(* PLC project LibIT, lamsystems-it.ru LibIT 1 *)
(* stored: creationDateTime 2019-11-13T09:37:45, productRelease 0, modificationDateTime 2022-04-28T12:46:30, version 0 *)

(* Increment of source value *)
FUNCTION Inc : INT
  VAR_INPUT
    Ex : BOOL;  (* execution allow *)
    V : INT;  (* source value *)
  END_VAR
  VAR
    Val : INT;
  END_VAR

            Val:= V;

IF Ex = True THEN
  Val:= V+1;
END_IF;

Inc:= Val;


          
END_FUNCTION

(* Decrement of source value *)
FUNCTION Dec : INT
  VAR_INPUT
    Ex : BOOL;  (* execution allow *)
    V : INT;  (* source value *)
  END_VAR
  VAR
    Val : INT;
  END_VAR

            Val:= V;

IF Ex = True AND Val > 0 THEN
  Val:= V-1;
END_IF;

Dec:= Val;


          
END_FUNCTION

(* Set bit value in source word *)
FUNCTION SetBitLWo : LWORD
  VAR_INPUT
    Wo : LWORD := 0;  (* source word *)
    Pos : BYTE := 0;  (* bit position (0..63) *)
    Val : BOOL := FALSE;  (* bit value *)
  END_VAR
  VAR
    Mask : LWORD := 0;
  END_VAR

            Mask:= REAL_TO_LWORD(EXPT(INT_TO_REAL(2),BYTE_TO_INT(Pos)));
IF Val = FALSE THEN
  SetBitLWo:= (Wo AND NOT(Mask));
ELSE
  SetBitLWo:= (Wo OR Mask);
END_IF;
          
END_FUNCTION

(* Get bit value from source word *)
FUNCTION GetBitLWo : BOOL
  VAR_INPUT
    Wo : LWORD := 0;  (* source word *)
    Pos : BYTE := 0;  (* bit position (0..63) *)
  END_VAR
  VAR
    Mask : LWORD := 0;
  END_VAR

            Mask:= REAL_TO_LWORD(EXPT(INT_TO_REAL(2),BYTE_TO_INT(Pos)));
GetBitLWo:= ((Wo AND Mask) > 0);

          
END_FUNCTION

(* Set bit value in source word *)
FUNCTION SetBitWo : WORD
  VAR_INPUT
    Wo : WORD := 0;  (* source word *)
    Pos : BYTE := 0;  (* bit position (0..15) *)
    Val : BOOL := FALSE;  (* bit value *)
  END_VAR
  VAR
    Mask : WORD := 0;
  END_VAR

            Mask:= REAL_TO_WORD(EXPT(INT_TO_REAL(2),BYTE_TO_INT(Pos)));
IF Val = FALSE THEN
  SetBitWo:= (Wo AND NOT(Mask));
ELSE
  SetBitWo:= (Wo OR Mask);
END_IF;
          
END_FUNCTION

(* Get bit value from source word *)
FUNCTION GetBitWo : BOOL
  VAR_INPUT
    Wo : WORD := 0;  (* source word *)
    Pos : BYTE := 0;  (* bit position (0..15) *)
  END_VAR
  VAR
    Mask : WORD := 0;
  END_VAR

            Mask:= REAL_TO_WORD(EXPT(INT_TO_REAL(2),BYTE_TO_INT(Pos)));
GetBitWo:= ((Wo AND Mask) > 0);

          
END_FUNCTION

(* Filtration of discrete value *)
FUNCTION_BLOCK FiltrD
  VAR_INPUT
    Ex : BOOL := FALSE;  (* execution allow *)
    V : BOOL := FALSE;  (* source value *)
    Tm : TIME := T#0ms;  (* filter delay (ms) *)
  END_VAR
  VAR_OUTPUT
    Ov : BOOL := FALSE;  (* filtered source value *)
  END_VAR
  VAR
    Val : BOOL := FALSE;
    TON0 : TON;
    TON1 : TON;
  END_VAR

            TON0(IN:=AND(Ex, NOT(V)), PT:=Tm);
TON1(IN:=AND(Ex, V), PT:=Tm);

IF TON0.Q = TRUE THEN
  Val:= FALSE;
END_IF;

IF TON1.Q = TRUE THEN
  Val:= TRUE;
END_IF;

Ov:= Val;

          
END_FUNCTION_BLOCK

(* Filtration of analog value *)
FUNCTION_BLOCK FiltrA
  VAR_INPUT
    Ex : BOOL := FALSE;  (* execution allow *)
    V : REAL := 0.0;  (* source value *)
    K : REAL := 0.0;  (* filter factor (0.0 .. 1.0) *)
  END_VAR
  VAR_OUTPUT
    Ov : REAL := 0.0;  (* filtered source value *)
  END_VAR
  VAR
    Val : REAL := 0.0;  (* stored value *)
    Klim : REAL := 0.0;  (* stored value *)
  END_VAR

            IF Ex = TRUE THEN
  Klim:= LIMIT(MN:=0.0, IN:=K, MX:=1.0);
  Val := (Klim*V)+(1.0-Klim)*Ov;
ELSE
  Val:= V;
END_IF;

Ov:= Val;

          
END_FUNCTION_BLOCK

(* Calculate scale angle factor *)
FUNCTION ScaleA_Ka : REAL
  VAR_INPUT
    Ex : BOOL := FALSE;  (* execution allow *)
    V1 : REAL := 0.0;  (* value of low point *)
    V2 : REAL := 0.0;  (* value of high point *)
    Y1 : REAL := 0.0;  (* calibration value of low point *)
    Y2 : REAL := 0.0;  (* calibration value of high point *)
    Ka : REAL := 0.0;  (* source value of the factor *)
  END_VAR

            IF Ex = TRUE THEN
  ScaleA_Ka:= (Y2-Y1)/(V2-V1);
ELSE  
  ScaleA_Ka:= Ka;
END_IF;

          
END_FUNCTION

(* Calculate scale offset factor *)
FUNCTION ScaleA_Kb : REAL
  VAR_INPUT
    Ex : BOOL := FALSE;  (* execution allow *)
    V1 : REAL := 0.0;  (* value of low point *)
    V2 : REAL := 0.0;  (* value of high point *)
    Y1 : REAL := 0.0;  (* calibration value of low point *)
    Y2 : REAL := 0.0;  (* calibration value of high point *)
    Kb : REAL := 0.0;  (* source value of the factor *)
  END_VAR

            IF Ex = TRUE THEN
  ScaleA_Kb:= ((Y1*V2)-(Y2*V1))/(V2-V1);
ELSE  
  ScaleA_Kb:= Kb;
END_IF;

          
END_FUNCTION

(* Scale of analog value *)
FUNCTION ScaleA : REAL
  VAR_INPUT
    Ex : BOOL := FALSE;  (* execution allow *)
    V : REAL := 0.0;  (* value of curent point *)
    Ka : REAL := 0.0;  (* angle factor *)
    Kb : REAL := 0.0;  (* offset factor *)
    Y : REAL := 0.0;  (* source scale value *)
  END_VAR

            IF Ex = TRUE THEN
  ScaleA:= (Ka*V)+Kb;
ELSE  
  ScaleA:= Y;
END_IF;

          
END_FUNCTION

(* Continuous TON *)
FUNCTION_BLOCK TONcont
  VAR_INPUT
    IN : BOOL := FALSE;  (* start command *)
  END_VAR
  VAR_OUTPUT
    Q : BOOL := FALSE;  (* status *)
    ET : TIME := T#0ms;  (* estimated time *)
  END_VAR
  VAR
    TON1 : TON;
    TON1_IN : BOOL := FALSE;
    TON1_TM : TIME := T#600000ms;
    TON1Inc : TON;
    TON1Inc_IN : BOOL := FALSE;
    TON1Inc_TM : TIME := T#300000ms;
  END_VAR

            TON1_IN   := IN;
TON1Inc_IN:= IN;

IF TON1Inc.Q = TRUE THEN
  TON1_TM   := ADD_TIME(IN1:=TON1_TM, IN2:=TON1Inc_TM);
  TON1Inc_IN:= FALSE;
END_IF;

TON1(IN:=TON1_IN, PT:=TON1_TM);
TON1Inc(IN:=TON1Inc_IN, PT:=TON1Inc_TM);

Q := TON1.Q;
ET:= TON1.ET;

          
END_FUNCTION_BLOCK

(* Autotuning of PID-controller *)
FUNCTION_BLOCK PIDtun
  VAR_INPUT
    Ex : BOOL := FALSE;  (* execution allow *)
    V : REAL := 0.0;  (* source value *)
    Diff : REAL := 0.0;  (* difference setpoint *)
    Ty : BYTE := 0;  (* type of controller *)
    Pro : BYTE := 0;  (* type of process *)
  END_VAR
  VAR_OUTPUT
    Ok : BYTE := 0;  (* result code *)
    OY : REAL := 0.0;  (* regulator value *)
    OKp : REAL := 0.0;  (* P-factor *)
    OKi : REAL := 0.0;  (* I-factor *)
    OKd : REAL := 0.0;  (* D-factor *)
    OTm : DWORD := 0;  (* cycle time (ms) *)
  END_VAR
  VAR
    OTmLocal : DWORD := 0;  (* cycle time (ms) *)
  END_VAR
  VAR_OUTPUT
    dETm : DWORD := 0;  (* error break control time (ms) *)
  END_VAR
  VAR
    dETmLocal : DWORD := 0;  (* error break control time (ms) *)
  END_VAR
  VAR_OUTPUT
    dE : REAL := 0.0;  (* dE value *)
  END_VAR
  VAR
    dELocal : REAL := 0.0;  (* dE value *)
    TunDone : BOOL := FALSE;
    Tm1 : REAL := 0.0;  (* t0 (ms) *)
    Tm2 : REAL := 0.0;  (* tu (ms) *)
    TmSum : REAL := 0.0;  (* t (ms) *)
    V1Set : BOOL := FALSE;
    V01 : REAL := 0.0;
    V063 : REAL := 0.0;
    Rr : REAL := 0.0;  (* R *)
    Tm1sec : REAL := 0.0;  (* t0 div 100 *)
    TONcont1 : TONcont;
    TONcont1_IN : BOOL := FALSE;
    CntChangeInVal : UINT := 0;
    StartVal : REAL := 0.0;
    PrewVal : REAL := 0.0;
  END_VAR

            (* Ty - regulator type *)
(* = 0 - PID *)
(* = 1 - PI *)
(* = 2 - PD *)
(* = 3 - P *)

(* Pro - process type *)
(* = 0 - increasing (by default) *)
(* = 1 - decreasing *)

(* Ok - result code *)
(* = 0 - off *)
(* = 1 - work *)
(* = 2 - incorrect regulator type *)
(* = 3 - work done success *)

IF Ex = TRUE THEN
  
  IF Ty <= 3 THEN
      
    IF TunDone = FALSE THEN
      
      (* work *)
      Ok:= 1;
      
      IF V1Set = FALSE THEN
        V1Set:= TRUE;
        CntChangeInVal:= 0;
        StartVal:= V;
        PrewVal:= V;        
        (* calculate setpoint for V(0.1) by type of process *)
        IF Pro = 1 THEN
          (* decreasing *)
          V01 := (V-(0.1*Diff));
          V063:= (V-(0.63*Diff));
        ELSE
          (* increasing *)
          V01 := (V+(0.1*Diff));
          V063:= (V+(0.63*Diff));
        END_IF;
      END_IF;
      
      (* set Tm1 (ms) *)
      IF V < V01 THEN
        Tm1:= TIME_TO_REAL(TONcont1.ET)*1000.0;
      END_IF;
      
      (* set Tm2 (ms) *)
      IF V >= V063 THEN
        
        TONcont1_IN:= FALSE;
        TunDone    := TRUE;
        
        Tm2   := TIME_TO_REAL(TONcont1.ET)*1000.0;
        TmSum := (Tm1+Tm2);
        (*OTm   := REAL_TO_DWORD((Tm1*1.875));*)
        Rr    := (Diff/((TmSum-Tm1)/1000.0));
        Tm1sec:= (Tm1/1000.0);
        (* 1000 - divider to convert msec to sec *)
        
        OTm:= OTmLocal; 
        dE:=dELocal;
        dETm:=dETmLocal;                
          
        (* calculate factors by type of regulator *)
        CASE BYTE_TO_INT(Ty) OF
          0:
            (* PID *)
            OKp:= (1.2/(Rr*Tm1sec));
            OKi:= (2.0*Tm1sec);
            OKd:= (0.4*Tm1sec);
          1:
            (* PI *)
            OKp:= (0.8/(Rr*Tm1sec));
            OKi:= (2.0*Tm1sec);
          2:
            (*PD*)
            OKp:= (1.0/(Rr*Tm1sec));
            OKd:= (0.25*Tm1sec);
          3:
            (*P*)
            OKp:= (1.0/(Rr*Tm1sec));
        END_CASE;
        
      END_IF;
      (* end of Tm2 *)
    ELSE
      (* work done success *)
      Ok:= 3;
    END_IF;
    (* end of TunDone *)
  ELSE
    (* incorrect regulator type *)
    Ok:= 2;
  END_IF;
  (* end of Ty *)
ELSE
  (* off *)
  Ok:= 0;
END_IF;
(* end of Ex *)

(* work *)
IF Ok = 1 THEN
  OY         := 100.0;
  TONcont1_IN:= TRUE;
  
  IF CntChangeInVal < 4 THEN  
   IF Pro = 0 THEN (* increasing *)
    IF V > StartVal AND V > PrewVal THEN
      CntChangeInVal:= (CntChangeInVal + 1);
      PrewVal:= V;
    (*ELSE*)
      (*CntChangeInVal:= 0;*)
    END_IF;
   ELSE (* decreasing *)
    IF V < StartVal AND V < PrewVal THEN
      CntChangeInVal:= (CntChangeInVal + 1);
      PrewVal:= V;
    (*ELSE*)
      (*CntChangeInVal:= 0;*)  
    END_IF;   
   END_IF;  
    (*PrewVal:= V;*)  
  END_IF;
  
  IF CntChangeInVal=4 THEN
   OTmLocal:= REAL_TO_DWORD(Tm1); 
   dELocal:=(PrewVal-StartVal);
   dETmLocal:=DINT_TO_DWORD((DWORD_TO_DINT(OTmLocal)*3));
   CntChangeInVal:= 5; 
  END_IF;   
  
END_IF;

(* off, error *)
IF Ok = 0 OR Ok = 2 THEN
  OY         := 0.0;
  TONcont1_IN:= FALSE;
  V1Set      := FALSE;
  TunDone    := FALSE;
  OKp        := 0.0;
  OKi        := 0.0;
  OKd        := 0.0;
  OTm        := 0;
  
  CntChangeInVal:= 0;
  StartVal:= 0.0;
  PrewVal:= 0.0;  
  
  OTmLocal:= 0; 
  dELocal:=0.0;
  dETmLocal:=0;  
  
  OTm:= 0; 
  dE:=0.0;
  dETm:=0;   
  
END_IF;

(* work is done success *)
IF TunDone = TRUE THEN
  OY         := 0.0;
END_IF;

TONcont1(IN:=TONcont1_IN);

(* DEBUG *)
(* set Class of debug variables to Output to use its as Outputs of the FB *)
(* set Class of debug variables to Local to hide its *)
(* Deb_V1 := V01; *)
(* Deb_Tm1:= Tm1; *)
(* Deb_V2 := V063; *)
(* Deb_Tm2:= Tm2; *)
(* end of DEBUG *)

          
END_FUNCTION_BLOCK

(* PID-controller (v1) *)
FUNCTION_BLOCK PID1
  VAR_INPUT
    Ex : BOOL := FALSE;  (* execution allow *)
    V : REAL := 0.0;  (* source value *)
    Sp : REAL := 0.0;  (* setpoint *)
    Ty : BYTE := 0;  (* type of controller *)
    Pro : BYTE := 0;  (* type of process *)
    Kp : REAL := 0.0;  (* P-factor *)
    Ki : REAL := 0.0;  (* I-factor *)
    Kd : REAL := 0.0;  (* D-factor *)
    Sck : BOOL := FALSE;  (* external command to start regulator cycle *)
    dI : REAL := 0.0;  (* integral zone *)
    dZ : REAL := 0.0;  (* dead zone *)
    dE : REAL := 0.0;  (* control failure zone *)
    dETm : DWORD := 5000;  (* control failure zone (time to detect zone, ms) *)
    Ym : BYTE := 0;  (* type of OY *)
  END_VAR
  VAR_OUTPUT
    Ok : BYTE := 0;  (* result code *)
    OY : REAL := 0.0;  (* regulator value (%) *)
  END_VAR
  VAR
    Er : REAL := 0.0;  (* error delta *)
    ErAbs : REAL := 0.0;  (* error delta (absolute) *)
    ErPrev : REAL := 0.0;  (* error delta (previous cycle) *)
    ErDiff : REAL := 0.0;  (* error delta (diff) *)
    Ppart : REAL := 0.0;  (* P-part *)
    Ipart : REAL := 0.0;  (* I-part *)
    Dpart : REAL := 0.0;  (* D-part *)
    DeV : REAL := 0.0;  (* control failure zone (1-point) *)
    DeV1Set : BOOL := FALSE;  (* control failure zone (1-point is set) *)
    DeV2Set : BOOL := FALSE;  (* control failure zone (2-point is set) *)
    SckSet : BOOL := FALSE;  (* external start (set) *)
    ErrorSet : BOOL := FALSE;  (* e-zone (set) *)
    TON_De : TON;
    TON_De_IN : BOOL := FALSE;
    TON_De_TM : TIME := T#0ms;
  END_VAR

            (* Ty - regulator type *)
(* = 0 - PID *)
(* = 1 - PI *)
(* = 2 - PD *)
(* = 3 - P *)

(* Pro - process type *)
(* = 0 - increasing (by default) *)
(* = 1 - decreasing *)

(* Ym - type of OY *)
(* = 0 - unipolar    0.0 .. 100.0 % (by default) *)
(* = 1 - bipolar  -100.0 .. 100.0 % *)

(* Ok - result code *)
(* = 0 - off *)
(* = 1 - work *)
(* = 2 - dead (d-)zone *)
(* = 3 - integral (i-)zone *)
(* = 4 - control failure (e-)zone *)
(* = 5 - incorrect regulator type *)

(* reset Sck *)
IF Sck = FALSE THEN
  SckSet:= FALSE;
END_IF;

(* test execution allow *)
IF Ex = TRUE THEN
  
  (* test regulator type *)
  IF Ty <= 3 THEN
    
    (* test start *)
    IF Sck = TRUE AND SckSet = FALSE AND ErrorSet = FALSE THEN
      
      SckSet:= TRUE;
      
      (* work *)
      Ok:= 1;
     
      Er    := (Sp-V);
      ErDiff:= (Er-ErPrev);
      ErPrev:= Er;
      ErAbs := ABS(IN:=Er);
      
      (* test d-zone *)
      IF ErAbs >= dZ THEN
        
        (* Ty: 0-PID, 1-PI, 2-PD, 3-P *)
        Ppart:= (Kp*Er);
        
        (* Ty: 0-PID, 1-PI *)
        IF (Ty = 0 OR Ty = 1) AND (ErAbs < dI OR dI = 0.0) AND Ki > 0.0 THEN
          (* i-zone *)
          Ok:= 3;
          Ipart:= (Ipart+Er);
          IF Ipart >= Ki THEN
            Ipart:= Ki;
          END_IF;
          Ipart:= ((1.0/Ki)*Ipart);
        ELSE
          Ipart:= 0.0;
        END_IF;
        
        (*0-PID, 2-PD*)
        IF (Ty = 0 OR Ty = 2) THEN
          Dpart:= (Kd*ErDiff);
        ELSE
          Dpart:= 0.0;
        END_IF;
        
        OY:= (Ppart+Ipart+Dpart)*100.0;
        
      ELSE
        (* d-zone *)
        Ok:= 2;
      END_IF;
      (* end of test d-zone *)
      
    END_IF;
    (* end of test start *)
  
  ELSE
    (* incorrect regulator type *)
    Ok:= 5;
    ErrorSet:= TRUE;
  END_IF;
  (* end of test regulator type *)
  
ELSE
  (* off *)
  Ok:= 0;
END_IF;
(* end of Ex *) 

(* work, i-zone *)
IF dETm >= 100 THEN  
 IF (Ok = 1 OR Ok = 3) AND ABS(IN:=OY) >= 100.0 THEN
    
  IF dETm > 0 THEN
    TON_De_TM:= REAL_TO_TIME(DWORD_TO_REAL(dETm)/1000.0);
    TON_De_IN:= TRUE;
  END_IF;
    
  IF DeV1Set = FALSE THEN
    (* point 1 *)
    DeV:= V;
    DeV1Set:= TRUE;
  END_IF;
    
  IF TON_De.Q = TRUE THEN
    IF DeV2Set = FALSE THEN
      (* point 2 *)
      DeV:= (V-DeV);
      DeV2Set:= TRUE;
    END_IF;
    IF DeV < dE OR DeV < 0.0 THEN
      (* e-zone *)
      Ok:= 4;
      ErrorSet:= TRUE;
    END_IF;
  END_IF;
  
 ELSE
  TON_De_IN:= FALSE;
  DeV1Set  := FALSE;
  DeV2Set  := FALSE;
 END_IF;
END_IF;

(* off *)
IF Ok = 0 THEN
  OY       := 0.0;
  SckSet   := FALSE;
  ErrorSet := FALSE;
  Ppart    := 0.0;
  Ipart    := 0.0;
  Dpart    := 0.0;
END_IF;

(* e-zone, error of regulator type *)
IF ErrorSet = TRUE THEN
  OY       := 0.0;
END_IF;

(* scale OY by type of process *)
IF Pro = 1 THEN
  (* decreasing *)
  OY:= (100.0-OY);
END_IF;

(* scale OY by type of output *)
IF Ym = 1 THEN
  (* bipolar *)
  OY:= LIMIT(MN:=-100.0, IN:=OY, MX:=100.0);
ELSE
  (* unipolar *)
  OY:= LIMIT(MN:=0.0, IN:=OY, MX:=100.0);
END_IF;

TON_De(IN:=TON_De_IN, PT:=TON_De_TM);

(* DEBUG *)
(* set Class of debug variables to Output to use its as Outputs of the FB *)
(* set Class of debug variables to Local to hide its *)
(* Deb_P   := Ppart; *)
(* Deb_I   := Ipart; *)
(* Deb_D   := Dpart; *)
(* Deb_dEEt:= REAL_TO_DWORD(TIME_TO_REAL(TON_De.ET)*1000.0); *)
(* end of DEBUG *)

          
END_FUNCTION_BLOCK

(* PID-controller (v2) *)
FUNCTION_BLOCK PID2
  VAR_INPUT
    Ex : BOOL := FALSE;  (* execution allow *)
    V : REAL := 0.0;  (* source value *)
    Sp : REAL := 0.0;  (* setpoint *)
    Ty : BYTE := 0;  (* type of controller *)
    Pro : BYTE := 0;  (* type of process *)
    Kp : REAL := 0.0;  (* P-factor *)
    Ki : REAL := 0.0;  (* I-factor *)
    Kd : REAL := 0.0;  (* D-factor *)
    Tm : DWORD := 1000;  (* cycle time (ms) *)
    dI : REAL := 0.0;  (* integral zone *)
    dZ : REAL := 0.0;  (* dead zone *)
    dE : REAL := 0.0;  (* control failure zone *)
    dETm : DWORD := 5000;  (* control failure zone (time to detect zone, ms) *)
    Ym : BYTE := 0;  (* type of OY *)
  END_VAR
  VAR_OUTPUT
    Ok : BYTE := 0;  (* result code *)
    OY : REAL := 0.0;  (* regulator value (%) *)
  END_VAR
  VAR
    TON_Work : TON;
    TON_Work_IN : BOOL := FALSE;
    TON_Work_TM : TIME := T#0ms;
    PID1_1 : PID1;
  END_VAR

            PID1_1(Ex:=Ex, V:=V, Sp:=Sp, Ty:=Ty, Pro:=Pro, Kp:=Kp, Ki:=Ki, Kd:=Kd, Sck:=TON_Work.Q, dI:=dI, dZ:=dZ, dE:=dE, dETm:=dETm, Ym:=Ym);

Ok:= PID1_1.Ok;
OY:= PID1_1.OY;

IF Ex = TRUE AND Tm > 0 THEN
  TON_Work_TM:= REAL_TO_TIME(DWORD_TO_REAL(Tm)/1000.0);
  TON_Work_IN:= TRUE;
ELSE
  TON_Work_IN:= FALSE;
END_IF;

IF TON_Work.Q = TRUE THEN
  TON_Work_IN:= FALSE;
END_IF;

TON_Work(IN:=TON_Work_IN, PT:=TON_Work_TM);

(* DEBUG *)
(* set Class of debug variables to Output to use its as Outputs of the FB *)
(* set Class of debug variables to Local to hide its *)
(* Deb_P   := PID1_1.Deb_P; *)
(* Deb_I   := PID1_1.Deb_I; *)
(* Deb_D   := PID1_1.Deb_D; *)
(* Deb_Et  := REAL_TO_DWORD(TIME_TO_REAL(TON_Work.ET)*1000.0); *)
(* Deb_dEEt:= PID1_1.Deb_dEEt; *)
(* end of DEBUG *)

          
END_FUNCTION_BLOCK

(* Test TON *)
FUNCTION_BLOCK TONtest
  VAR_INPUT
    IN : BOOL := FALSE;  (* start command *)
    MS : DWORD := 0;  (* counter reference (msec) *)
  END_VAR
  VAR_OUTPUT
    Q : BOOL := FALSE;  (* status *)
    ET : TIME := T#0ms;  (* counter value (msec) *)
    EDW : DWORD := 0;  (* counter value (msec) *)
    EREA : REAL := 0.0;
  END_VAR
  VAR
    TON1 : TON;
    TON1_IN : BOOL := FALSE;
    TON1_TM : TIME := T#0ms;
  END_VAR

            TON1_IN:= IN;
TON1_TM:= REAL_TO_TIME(DWORD_TO_REAL(MS)/1000.0);

TON1(IN:=TON1_IN, PT:=TON1_TM);
Q   := TON1.Q;
ET  := TON1.ET;
EDW := REAL_TO_DWORD(TIME_TO_REAL(TON1.ET)*1000.0);
EREA:= TIME_TO_REAL(TON1.ET);
          
END_FUNCTION_BLOCK

FUNCTION_BLOCK FLR1
  VAR_INPUT
    Ex : BOOL := FALSE;  (* execution allow *)
    OrdInp : BOOL := TRUE;  (* order input value (0 - first order 1 - second or more order) *)
    V : REAL := 0.0;  (* source value *)
    Sp : REAL := 0.0;  (* setpoint *)
    StartOY : REAL := 0.0;  (* Start regulator value (%) *)
    Pro : BYTE := 0;  (* type of process *)
    Sck : BOOL := FALSE;  (* external command to start regulator cycle *)
    Tm : DWORD := 0;  (* cycle time (ms) *)
    dV : REAL := 0.0;  (* increment step of OY (%) *)
    dZ : REAL := 0.0;  (* dead zone *)
    dE : REAL := 0.0;  (* control failure zone *)
    dETm : DWORD := 5000;  (* control failure zone (time to detect zone, ms) *)
    Ym : BYTE := 0;  (* type of OY *)
  END_VAR
  VAR_OUTPUT
    Ok : BYTE := 0;  (* result code *)
    OY : REAL := 0.0;  (* regulator value (%) *)
  END_VAR
  VAR
    Vprev : REAL := 0.0;  (* previous source value *)
    TmDv : REAL := 0.0;  (* dV time (ms) *)
    UpDown : SINT := 0;  (* flag UpDown *)
    SckSet : BOOL := FALSE;  (* external start (set) *)
    ErrorSet : BOOL := FALSE;  (* e-zone (set) *)
    Er : REAL := 0.0;  (* error delta *)
    TON_De : TON;
    TON_De_IN : BOOL := FALSE;
    TON_De_TM : TIME := T#0ms;
    DeV : REAL := 0.0;  (* control failure zone (1-point) *)
    DeV1Set : BOOL := FALSE;  (* control failure zone (1-point is set) *)
    DeV2Set : BOOL := FALSE;  (* control failure zone (2-point is set) *)
    TON_Dv : TON;
    TON_Dv_IN : BOOL := FALSE;
    TON_Dv_TM : TIME := T#0ms;
  END_VAR

            (* Pro - process type *)
(* = 0 - increasing (by default) *)
(* = 1 - decreasing *)

(* Ym - type of OY *)
(* = 0 - unipolar    0.0 .. 100.0 % (by default) *)
(* = 1 - bipolar  -100.0 .. 100.0 % *)

(* Ok - result code *)
(* = 0 - off *)
(* = 1 - work *)
(* = 2 - dead (d-)zone *)
(* = 4 - control failure (e-)zone *)

(* reset Sck *)
IF Sck = FALSE THEN
  SckSet:= FALSE;
END_IF;

(* test execution allow *)
IF Ex = TRUE THEN
    
  (* test start *)
  IF Sck = TRUE AND SckSet = FALSE AND ErrorSet = FALSE THEN
    
    SckSet:= TRUE;  
    
    IF Ok = 0 THEN
      OY:= StartOY;
    END_IF;
          
    (* work *)
    Ok:= 1;
    
    Er:= (Sp-V);
    
    (* test d-zone *)
    IF ABS(IN:=Er) >= dZ THEN
      (* exec *)
      {extern void AppFlr(FLR1*);AppFlr(data__);}
    ELSE
      (* d-zone *)
      Ok:= 2;
    END_IF;
    (* end of test d-zone *)
      
  END_IF;
  (* end of test start *)
  
ELSE
  (* off *)
  Ok:= 0;
END_IF;
(* end of Ex *) 

(* work *)
IF Ok = 1 THEN
  
  IF TmDv > 0.0 THEN
    (* msec to real-sec to time *)
    TON_Dv_TM:= REAL_TO_TIME(TmDv/1000.0);
    TON_Dv_IN:= TRUE;
  END_IF;
  
  IF TON_Dv.Q = TRUE THEN
    TON_Dv_IN:= FALSE;
    (* down *)
    IF UpDown = -1 THEN
      OY:= OY-dV;
    END_IF;
    (* up *)
    IF UpDown = 1 THEN
      OY:= OY+dV;
    END_IF;
  END_IF;
  
ELSE
  TON_Dv_IN:= FALSE;
END_IF;
(* end of work *)

(* test e-zone *)
IF dETm >= 100 THEN  
 IF Ok = 1 AND ABS(IN:=OY) >= 100.0 THEN
  
  IF dETm > 0 THEN
    (* msec to real-sec to time *)
    TON_De_TM:= REAL_TO_TIME(DWORD_TO_REAL(dETm)/1000.0);
    TON_De_IN:= TRUE;
  END_IF;
    
  IF DeV1Set = FALSE THEN
    (* point 1 *)
    DeV:= V;
    DeV1Set:= TRUE;
  END_IF;
    
  IF TON_De.Q = TRUE THEN
    IF DeV2Set = FALSE THEN
      (* point 2 *)
      DeV:= (V-DeV);
      DeV2Set:= TRUE;
    END_IF;
    IF DeV < dE OR DeV < 0.0 THEN
      (* e-zone *)
      Ok:= 4;
      ErrorSet:= TRUE;
    END_IF;
  END_IF;
  
 ELSE
  TON_De_IN:= FALSE;
  DeV1Set  := FALSE;
  DeV2Set  := FALSE;
 END_IF;
END_IF;
(* end of test e-zone *)

(* off *)
IF Ok = 0 THEN
  OY       := 0.0;
  SckSet   := FALSE;
  ErrorSet := FALSE;
  Vprev    := 0.0;
END_IF;

(* error *)
IF ErrorSet = TRUE THEN
  OY       := 0.0;
END_IF;

(* scale OY by type of process *)
IF Pro = 1 THEN
  (* decreasing *)
  OY:= (100.0-OY);
END_IF;


(* work *)
IF Ok = 1 THEN
  (* scale OY by type of output *)
  IF Ym = 1 THEN
    (* bipolar *)
    OY:= LIMIT(MN:=-100.0, IN:=OY, MX:=100.0);
  ELSE
    (* unipolar *)
    OY:= LIMIT(MN:=0.0, IN:=OY, MX:=100.0);
  END_IF;
END_IF;

TON_De(IN:=TON_De_IN, PT:=TON_De_TM);
TON_Dv(IN:=TON_Dv_IN, PT:=TON_Dv_TM);

(* DEBUG *)
(* set Class of debug variables to Output to use its as Outputs of the FB *)
(* set Class of debug variables to Local to hide its *)
(* Deb_UpDown:= UpDown; *)
(* Deb_dVTm  := REAL_TO_DWORD(TmDv); *)
(* Deb_dVEt  := REAL_TO_DWORD(TIME_TO_REAL(TON_Dv.ET)*1000.0); *)
(* Deb_dEEt  := REAL_TO_DWORD(TIME_TO_REAL(TON_De.ET)*1000.0); *)
(* end of DEBUG *)

          
END_FUNCTION_BLOCK

FUNCTION_BLOCK FLR2
  VAR_INPUT
    Ex : BOOL := FALSE;  (* execution allow *)
    OrdInp : BOOL := TRUE;  (* order input value (0 - first order 1 - second or more order) *)
    V : REAL := 0.0;  (* source value *)
    Sp : REAL := 0.0;  (* setpoint *)
    StartOY : REAL := 0.0;  (* Start regulator value (%) *)
    Pro : BYTE := 0;  (* type of process *)
    Tm : DWORD := 0;  (* cycle time (ms) *)
    dV : REAL := 0.0;  (* increment step of OY (%) *)
    dZ : REAL := 0.0;  (* dead zone *)
    dE : REAL := 0.0;  (* control failure zone *)
    dETm : DWORD := 5000;  (* control failure zone (time to detect zone, ms) *)
    Ym : BYTE := 0;  (* type of OY *)
  END_VAR
  VAR_OUTPUT
    Ok : BYTE := 0;  (* result code *)
    OY : REAL := 0.0;  (* regulator value (%) *)
  END_VAR
  VAR
    TON_Work : TON;
    TON_Work_IN : BOOL := FALSE;
    TON_Work_TM : TIME := T#0ms;
    FLR1_1 : FLR1;
  END_VAR

            FLR1_1(Ex:=Ex, OrdInp:=OrdInp, V:=V, Sp:=Sp, StartOY:=StartOY, Pro:=Pro, Sck:=TON_Work.Q, Tm:=Tm, dV:=dV, dZ:=dZ, dE:=dE, dETm:=dETm, Ym:=Ym);

Ok:= FLR1_1.Ok;
OY:= FLR1_1.OY;

IF Ex = TRUE AND Tm > 0 THEN
  (* msec to real-sec to time *)
  TON_Work_TM:= REAL_TO_TIME(DWORD_TO_REAL(Tm)/1000.0);
  TON_Work_IN:= TRUE;
ELSE
  TON_Work_IN:= FALSE;
END_IF;

IF TON_Work.Q = TRUE THEN
  TON_Work_IN:= FALSE;
END_IF;

TON_Work(IN:=TON_Work_IN, PT:=TON_Work_TM);

(* DEBUG *)
(* set Class of debug variables to Output to use its as Outputs of the FB *)
(* set Class of debug variables to Local to hide its *)
(* Deb_Speed := FLR1_1.Deb_Speed; *)
(* Deb_UpDown:= FLR1_1.Deb_UpDown; *)
(* Deb_dVTm  := FLR1_1.Deb_dVTm; *)
(* Deb_dVEt  := FLR1_1.Deb_dVEt; *)
(* Deb_dEEt  := FLR1_1.Deb_dEEt; *)
(* Deb_Et    := REAL_TO_DWORD(TIME_TO_REAL(TON_Work.ET)*1000.0); *)
(* Deb_Y0    := FLR1_1.Deb_Y0; *)
(* Deb_Er    := FLR1_1.Deb_Er; *)
(* Deb_Cm    := FLR1_1.Deb_Cm; *)
(* Deb_m     := FLR1_1.Deb_m; *)
(* end of DEBUG *)

          
END_FUNCTION_BLOCK

(* Autotuning of FLR-controller *)
FUNCTION_BLOCK FLRtun
  VAR_INPUT
    Ex : BOOL := FALSE;  (* execution allow *)
    V : REAL := 0.0;  (* source value *)
    Diff : REAL := 0.0;  (* difference setpoint *)
    Pro : BYTE := 0;  (* type of process *)
  END_VAR
  VAR_OUTPUT
    Ok : BYTE := 0;  (* result code *)
    OY : REAL := 0.0;  (* regulator value *)
    OTm : DWORD := 0;  (* cycle time (ms) *)
  END_VAR
  VAR
    OTmLocal : DWORD := 0;  (* cycle time (ms) *)
  END_VAR
  VAR_OUTPUT
    dETm : DWORD := 0;  (* error break control time (ms) *)
  END_VAR
  VAR
    dETmLocal : DWORD := 0;  (* error break control time (ms) *)
  END_VAR
  VAR_OUTPUT
    dE : REAL := 0.0;  (* dE value *)
  END_VAR
  VAR
    dELocal : REAL := 0.0;  (* dE value *)
    TunDone : BOOL := FALSE;
    Tm1 : REAL := 0.0;  (* t0 (ms) *)
    V1Set : BOOL := FALSE;
    V01 : REAL := 0.0;
    TONcont1 : TONcont;
    TONcont1_IN : BOOL := FALSE;
    CntChangeInVal : UINT := 0;
    StartVal : REAL := 0.0;
    PrewVal : REAL := 0.0;
  END_VAR

            (* Pro - process type *)
(* = 0 - increasing (by default) *)
(* = 1 - decreasing *)

(* Ok - result code *)
(* = 0 - off *)
(* = 1 - work *)
(* = 3 - work done success *)

IF Ex = TRUE THEN
  
  IF TunDone = FALSE THEN
      
    (* work *)
    Ok:= 1;
      
    IF V1Set = FALSE THEN
      V1Set:= TRUE;
      CntChangeInVal:= 0;
      StartVal:= V;
      PrewVal:= V;
      (* calculate setpoint for V(0.1) by type of process *)
      IF Pro = 1 THEN
        (* decreasing *)
        V01 := (V-(0.1*Diff));
      ELSE
        (* increasing *)
        V01 := (V+(0.1*Diff));
      END_IF;
    END_IF;
      
    (* set Tm1 (ms) *)
    IF V < V01 THEN
      Tm1:= TIME_TO_REAL(TONcont1.ET)*1000.0;
    ELSE
      IF CntChangeInVal=5 THEN 
        (*OTm:= REAL_TO_DWORD((Tm1*1.875));*)
        OTm:= OTmLocal; 
        dE:=dELocal;
        dETm:=dETmLocal;        
        TunDone:= TRUE;
        (* work done success *)
        Ok:= 3;
      END_IF;  
    END_IF;
    
  END_IF;
  (* end of TunDone *)
    
ELSE
  (* off *)
  Ok:= 0;
END_IF;
(* end of Ex *)

(* work *)
IF Ok = 1 THEN
  OY         := 100.0;
  TONcont1_IN:= TRUE;

  IF CntChangeInVal < 4 THEN  
   IF Pro = 0 THEN (* increasing *)
    IF V > StartVal AND V > PrewVal THEN
      CntChangeInVal:= (CntChangeInVal + 1);
      PrewVal:= V;
    (*ELSE*)
      (*CntChangeInVal:= 0;*)  
    END_IF;
   ELSE (* decreasing *)
    IF V < StartVal AND V < PrewVal THEN
      CntChangeInVal:= (CntChangeInVal + 1);
      PrewVal:= V;
    (*ELSE*)
      (*CntChangeInVal:= 0;*)
    END_IF;   
   END_IF;  
      
  END_IF;
  
  IF CntChangeInVal=4 THEN
   OTmLocal:= REAL_TO_DWORD(Tm1); 
   dELocal:=(PrewVal-StartVal);
   dETmLocal:=DINT_TO_DWORD((DWORD_TO_DINT(OTmLocal)*3));
   CntChangeInVal:= 5; 
  END_IF;  
  
END_IF;

(* off, error *)
IF Ok = 0 THEN
  OY         := 0.0;
  TONcont1_IN:= FALSE;
  V1Set      := FALSE;
  TunDone    := FALSE;
  OTm        := 0;
  
  CntChangeInVal:= 0;
  StartVal:= 0.0;
  PrewVal:= 0.0;  
  
  OTmLocal:= 0; 
  dELocal:=0.0;
  dETmLocal:=0;  
  
  OTm:= 0; 
  dE:=0.0;
  dETm:=0;  
END_IF;

(* work is done success *)
IF TunDone = TRUE THEN
  OY         := 0.0;
  TONcont1_IN:= FALSE;
END_IF;

TONcont1(IN:=TONcont1_IN);

(* DEBUG *)
(* set Class of debug variables to Output to use its as Outputs of the FB *)
(* set Class of debug variables to Local to hide its *)
(* Deb_V1 := V01; *)
(* Deb_Tm1:= Tm1; *)
(* end of DEBUG *)

          
END_FUNCTION_BLOCK
